// TIA Portal V20 export
// export: Created 2025-12-01T14:57:05.5956146Z, ExportSetting None, DisplayName Totally Integrated Automation Portal, DisplayVersion V20 Update 3, DisplayName TIA Portal Openness, DisplayVersion V20 Update 3, DisplayName TIA Portal Version Control Interface, DisplayVersion V20 Update 3, DisplayName STEP 7 Professional, DisplayVersion V20 Update 3, DisplayName STEP 7 Safety, DisplayVersion V20 Update 2, DisplayName WinCC Basic/Comfort/Advanced, DisplayVersion V20 Update 3, DisplayName WinCC Professional, DisplayVersion V20 Update 3, DisplayName WinCC Unified, DisplayVersion V20 Update 3
FUNCTION "FC870_MesaSinUT" : Void   // FC870, LAD
TITLE = "MesaSinUT"
{ S7_Optimized_Access := 'FALSE' }
AUTHOR : TRACKING
NAME : 20130301
VERSION : 3.0
// Devuelve si hay UT o no en la Mesa (bool)
// stored: AutoNumber false, SetENOAutomatically false
   VAR_INPUT
      Mesa : UInt;   // Mesa que se quiere ver si no hay UT's
   END_VAR
   VAR_OUTPUT
      SinUT : Bool;   // La Mesa no tiene UT
   END_VAR
   VAR_TEMP
      Relleno : Byte;
      ValorReturn : Int;
   END_VAR
BEGIN

NETWORK
TITLE = Inicializar
////////////////////////////////////////////////////////////////////////////
// --- Reseteo Variable de Salida

      SET;
      =     #SinUT;  // Activo: No hay UT's



NETWORK
TITLE = Comprobar si hay UT en la Mesa
////////////////////////////////////////////////////////////////////////////
// --- Leer Cola de la Mesa


////////////////////////////////////////////////////////////////////////////
// --- Comprobacion de que la Mesa tenga UT o No

      L     "DB810_ColasMesas".Colas[#Mesa].UT_PrimeraMesa;
      L     0;
      ==I;
      JC    Final;  // No hay UT's ?

      CLR;
      =     #SinUT;  // Desactivo: Hay UT's

Final:NOP   0;  // Finalizar Funcion


END_FUNCTION
